// Mitsubishi GX Works2 project: q3   PLC: Q02/Q02H

PROGRAM MAIN
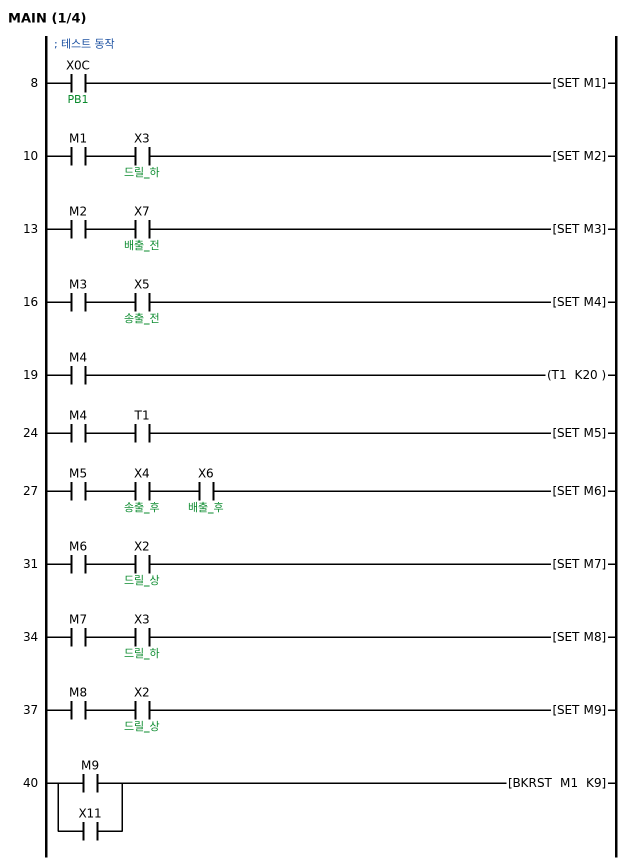
; 테스트 동작
8     LD      X0C  ; PB1
      SET     M1
10    LD      M1
      AND     X3  ; 드릴_하
      SET     M2
13    LD      M2
      AND     X7  ; 배출_전
      SET     M3
16    LD      M3
      AND     X5  ; 송출_전
      SET     M4
19    LD      M4
      OUT     T1 K20
24    LD      M4
      AND     T1
      SET     M5
27    LD      M5
      AND     X4  ; 송출_후
      AND     X6  ; 배출_후
      SET     M6
31    LD      M6
      AND     X2  ; 드릴_상
      SET     M7
34    LD      M7
      AND     X3  ; 드릴_하
      SET     M8
37    LD      M8
      AND     X2  ; 드릴_상
      SET     M9
40    LD      M9
      OR      X11
      BKRST   M1 K9
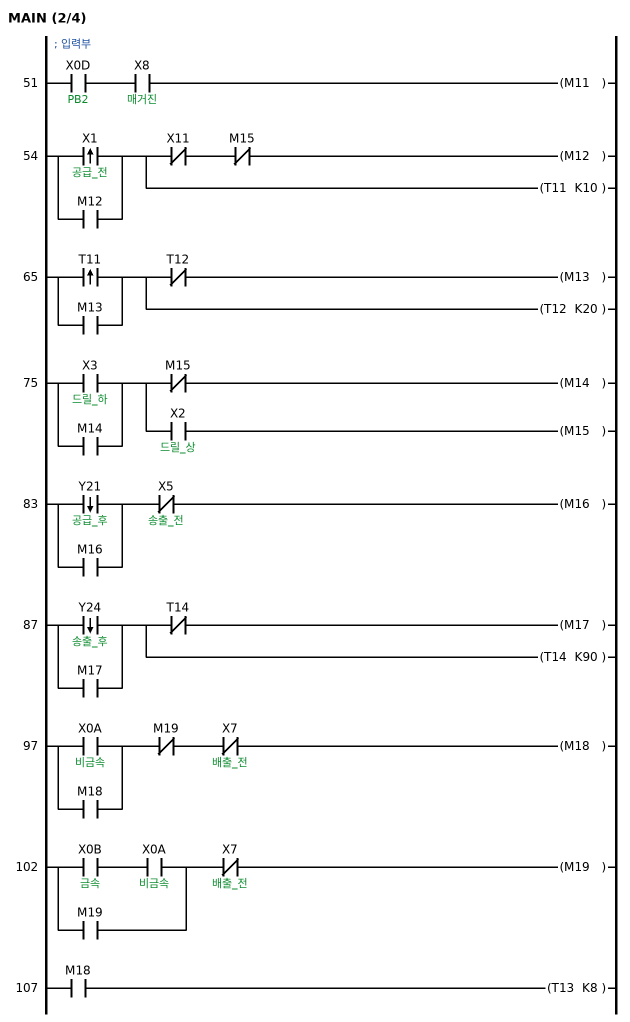
; 입력부
51    LD      X0D  ; PB2
      AND     X8  ; 매거진
      OUT     M11
54    LDP     X1  ; 공급_전
      OR      M12
      MPS
      ANI     X11
      ANI     M15
      OUT     M12
      MPP
      OUT     T11 K10
65    LDP     T11
      OR      M13
      MPS
      ANI     T12
      OUT     M13
      MPP
      OUT     T12 K20
75    LD      X3  ; 드릴_하
      OR      M14
      MPS
      ANI     M15
      OUT     M14
      MPP
      AND     X2  ; 드릴_상
      OUT     M15
83    LDF     Y21  ; 공급_후
      OR      M16
      ANI     X5  ; 송출_전
      OUT     M16
87    LDF     Y24  ; 송출_후
      OR      M17
      MPS
      ANI     T14
      OUT     M17
      MPP
      OUT     T14 K90
97    LD      X0A  ; 비금속
      OR      M18
      ANI     M19
      ANI     X7  ; 배출_전
      OUT     M18
102   LD      X0B  ; 금속
      AND     X0A  ; 비금속
      OR      M19
      ANI     X7  ; 배출_전
      OUT     M19
107   LD      M18
      OUT     T13 K8
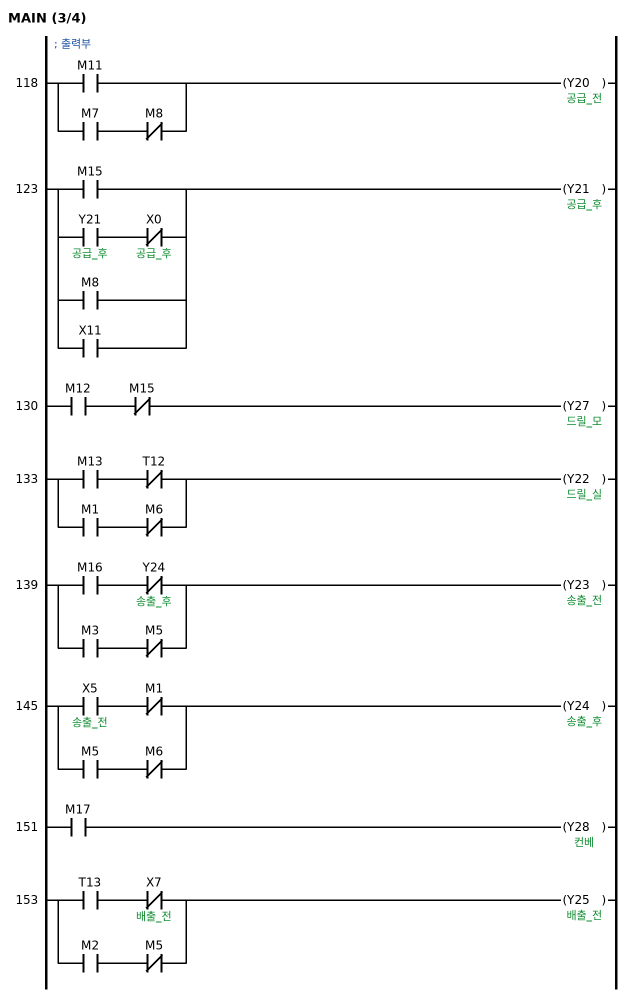
; 출력부
118   LD      M11
      LD      M7
      ANI     M8
      ORB
      OUT     Y20  ; 공급_전
123   LD      M15
      LD      Y21  ; 공급_후
      ANI     X0  ; 공급_후
      ORB
      OR      M8
      OR      X11
      OUT     Y21  ; 공급_후
130   LD      M12
      ANI     M15
      OUT     Y27  ; 드릴_모
133   LD      M13
      ANI     T12
      LD      M1
      ANI     M6
      ORB
      OUT     Y22  ; 드릴_실
139   LD      M16
      ANI     Y24  ; 송출_후
      LD      M3
      ANI     M5
      ORB
      OUT     Y23  ; 송출_전
145   LD      X5  ; 송출_전
      ANI     M1
      LD      M5
      ANI     M6
      ORB
      OUT     Y24  ; 송출_후
151   LD      M17
      OUT     Y28  ; 컨베
153   LD      T13
      ANI     X7  ; 배출_전
      LD      M2
      ANI     M5
      ORB
      OUT     Y25  ; 배출_전
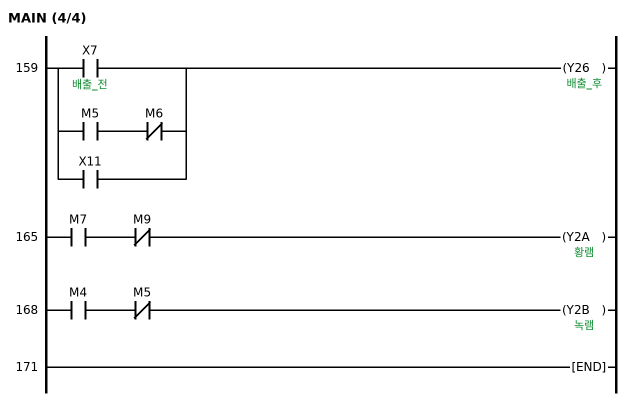
159   LD      X7  ; 배출_전
      LD      M5
      ANI     M6
      ORB
      OR      X11
      OUT     Y26  ; 배출_후
165   LD      M7
      ANI     M9
      OUT     Y2A  ; 황램
168   LD      M4
      ANI     M5
      OUT     Y2B  ; 녹램
171   END
END_PROGRAM

// device comments not shown above
X9  ; 이송감지
X0E  ; PB3
X0F  ; 비상정지
Y29  ; 적램
